PROGRAM Motor_move
VAR
	motorDirection_rotate: Motor_Direction;
	position_rotation: UINT;
	writeRotateReference: BOOL;
	writeHorizontalReference: BOOL;
	writeVerticalReference: BOOL;
	tolerance: UINT :=20;
	movemotor_rotate: Motor_Enable;
	desiredSpeed: INT :=5000;
END_VAR

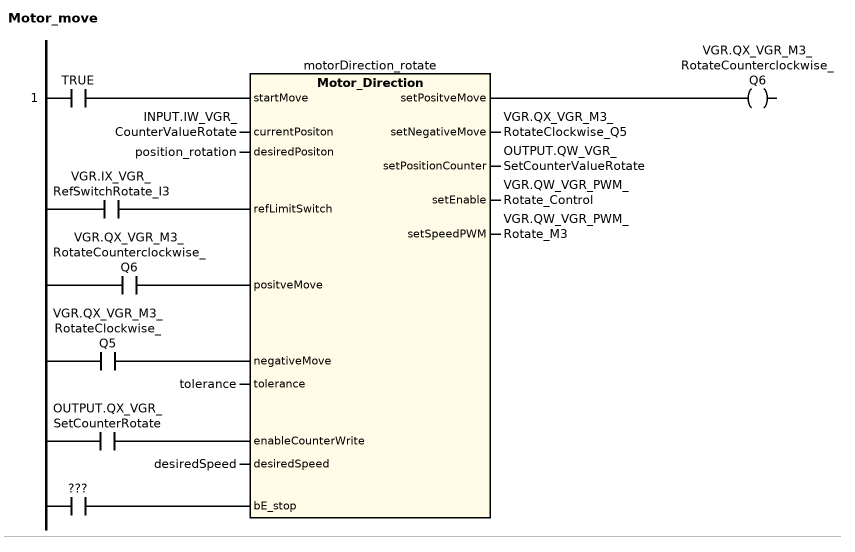
// NETWORK 1
motorDirection_rotate(
    startMove := TRUE,
    currentPositon := INPUT.IW_VGR_CounterValueRotate,
    desiredPositon := position_rotation,
    refLimitSwitch := VGR.IX_VGR_RefSwitchRotate_I3,
    positveMove := VGR.QX_VGR_M3_RotateCounterclockwise_Q6,
    negativeMove := VGR.QX_VGR_M3_RotateClockwise_Q5,
    tolerance := tolerance,
    enableCounterWrite := OUTPUT.QX_VGR_SetCounterRotate,
    desiredSpeed := desiredSpeed,
    setNegativeMove => VGR.QX_VGR_M3_RotateClockwise_Q5,
    setPositionCounter => OUTPUT.QW_VGR_SetCounterValueRotate,
    setEnable => VGR.QW_VGR_PWM_Rotate_Control,
    setSpeedPWM => VGR.QW_VGR_PWM_Rotate_M3); // Motor_Direction
VGR.QX_VGR_M3_RotateCounterclockwise_Q6 := motorDirection_rotate.setPositveMove;

END_PROGRAM

(* stored: Version 1.1.0.1, ProductVersion 3.1.4024.12
   POU Motor_move: Id {9a04db00-abe5-4125-8ad3-35cb329d63fd}, SpecialFunc None *)
